Fanuc KAREL source: ko00046.KL

-- PROVISIONAL review KL for V770-1; original PC SHA256 9f7f75075d347ea05f2b6d17385a5da8131aafcf3723d014ed8e0b9bffe77b32
-- Incomplete behavior may be omitted. Consult companion uncertainty JSON. Do not deploy.
PROGRAM KO00046
%NOLOCKGROUP
BEGIN
  -- UNRESOLVED_PC offsets 5-12; opcodes 9D,23
  -- UNRESOLVED_PC offsets 17-69; opcodes 27,27,49,7E,AD,27,49,7E,AD,22,31,7E,4A
  -- UNRESOLVED_PC offsets 74-78; opcodes 7F
END KO00046
